// TIA Portal V17 export
// export: Created 2022-12-01T11:06:40.0835024Z, ExportSetting WithDefaults, DisplayName Totally Integrated Automation Portal, DisplayVersion V17 Update 3, DisplayName TIA Portal Openness, DisplayVersion V17 Update 3, DisplayName TIA Portal Version Control Interface, DisplayVersion V17, DisplayName STEP 7 Professional, DisplayVersion V17 Update 3, DisplayName STEP 7 Safety, DisplayVersion V17, DisplayName WinCC Advanced, DisplayVersion V17 Update 3
FUNCTION "Gestion balizas" : Void   // FC1, STL
{ S7_Optimized_Access := 'TRUE' }
VERSION : 0.1
// stored: AutoNumber true, UDAEnableTagReadback false
   VAR_TEMP
      Report_Temp : "IFZ_Report";
      Word_Aux : Word;
      Entrada_Aux : Bool;
      Salida_Aux : Bool;
      Error_Aux : Bool;
      Reset_Aux : Bool;
      Rearme_PE_Blink : Bool;
      Sirena_Aux : Bool;
      Sirena_2_Aux : Bool;
      Sirena_3_Aux : Bool;
      Error_2_Aux : Bool;
      Error_3_Aux : Bool;
      Aire_Aux : Bool;
      Valor_Ant : Bool;
      Dint_Aux : DInt;
      Error_BLF1 : Bool;
      Error_BLF2 : Bool;
      Error_BLF3 : Bool;
      INSERTAR_REARME : Bool;
      Arrancando_Aux : Bool;
      INSERTAR_BALIZA : Bool;
      Paro_Instalacion_Aux : Bool;
      ZE_Pendiente_Rearme : Bool;
   END_VAR
BEGIN

NETWORK
TITLE = 
// Tras rearme de emergencias; el sistema, antes de arrancar, debe avisar mediante sirena (de los cuadros de control asociados a la zona de emergencia activada) de la siguiente forma: 5 segundos de forma intermitente (1Hz) y 3 segundos con sonido continuo. Tras este aviso de 8 segundos, el sistema arrancará normalmente.
      A     "Reset atascos";
      =     #Reset_Aux;

      CALL  "FC14_Balizas"
      ( Inicializar_Reporte := TRUE,
        Reset               := #Reset_Aux,
        Periferia           := FALSE,
        Emergencia          := #Report_Temp.F_Emergencia,
        F_Termico           := #Report_Temp.F_Termico,
        F_Atasco            := #Report_Temp.F_Atasco,
        F_Seccionador       := "Bit_basura",
        F_Galibo            := "Bit_basura",
        Manual              := #Report_Temp.Manual,
        Alimentacion        := #Report_Temp.F_Alimentacion,
        Alimentacion_CTR    := #Report_Temp.F_Alimentacion_CTR,
        Arrancando          := "Bit_basura",
        Pendiente_Rearme    := #Report_Temp.Pendiente_Rearme,
        Error               := #Error_Aux,
        Sirena              := #Sirena_Aux,
        CS_Error            := "Bit_basura",
        CS_Blink            := "Bit_basura",
        Report_Zona         := "DB1_Control".Z_R.Z_Proceso_1,
        Report_Global       := "DB1_Control".Z_R.Z_CC1,
        Control_Zona        := "DB1_Control".Z_C.Z_Proceso_1
      );

      A     #Error_Aux;
      AN    #Paro_Instalacion_Aux;
      =     "Baliza_PE";
      =     "Baliza_atasco";

      A     #Report_Temp.F_Emergencia;
      AN    #Paro_Instalacion_Aux;
      AN    #ZE_Pendiente_Rearme;
      =     "Baliza_atasco";
END_FUNCTION
